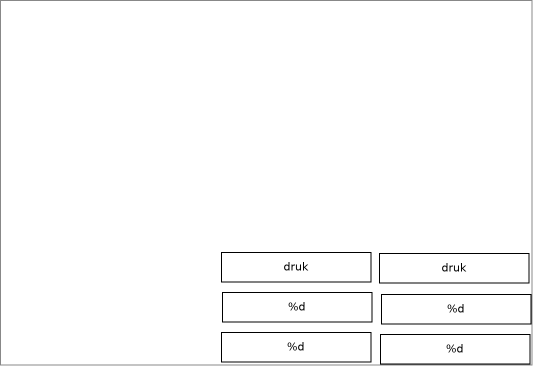
VISUALIZATION Visualization  // 533x366
    Rectangle (221,252 150x30), "druk", colour toggle: MAIN.lichten_1.lamp
        tap MAIN.vDruk_1
    Rectangle (379,253 150x30), "druk", colour toggle: MAIN.lichten_2.lamp
        tap MAIN.vDruk_2
    Rectangle (222,292 150x30), "%d", text variable: MAIN.LDR_1
    Rectangle (381,294 150x30), "%d", text variable: MAIN.LDR_2
    Rectangle (221,332 150x30), "%d", text variable: MAIN.LDR_3
    Rectangle (380,334 150x30), "%d", text variable: MAIN.LDR_4
END_VISUALIZATION

(* stored: Version 1.1.0.1, ProductVersion 3.1.4022.12
   Visu Visualization: Id {62db7a41-5546-4c87-ad92-cd947175c80c} *)
